// TwinCAT 3 PLC project PLC
// ProgramVersion: 3.1.4024.0
// libraries:
//   Tc2_Standard, * (Beckhoff Automation GmbH)
//   Tc2_System, * (Beckhoff Automation GmbH)
//   Tc3_Module, * (Beckhoff Automation GmbH)
// project tree:
//   / GlobalTextList.TcGTLO (not stored), PlcTask.TcTTO, VisualizationManager.TcVMO (not stored)
//   GVLs/ GVL.TcGVL (not stored)
//   POUs/ FB_VisuSim.TcPOU, MAIN.TcPOU (not stored), FB_StateMachine.TcPOU
//   VISUs/ Visu.TcVIS
// real-time tasks:
//   TASK PlcTask: cycle T#10ms, priority 20, ADS port 350
//   TASK VISU_TASK: cycle T#200000us, priority 30, ADS port 351

CONFIGURATION PLC
    RESOURCE PLC ON TwinCAT3
        TASK PlcTask(INTERVAL := T#10ms, PRIORITY := 20);
        PROGRAM MAIN WITH PlcTask : MAIN;
    END_RESOURCE
END_CONFIGURATION

// ---- POUs/FB_VisuSim.TcPOU
FUNCTION_BLOCK FB_VisuSim
VAR_INPUT
	bConveyor : BOOL;
END_VAR
VAR_OUTPUT
	bBottle : BOOL;
END_VAR
VAR
	fPos : REAL;
END_VAR

IF bConveyor THEN
	fPos := fPos + 0.1;
END_IF

IF fPos >= 100.0 THEN
	fPos := 0;
END_IF

bBottle := fPos >= 60.0 AND fPos <= 80.0;

END_FUNCTION_BLOCK

// ---- POUs/FB_StateMachine.TcPOU
(* -----------------------------------------------------------------------------
| This sample has been supplied by Beckhoff As-Is and is intended only as an   |
| example implementation. Functionality is not guaranteed.                     |
----------------------------------------------------------------------------- *)

FUNCTION_BLOCK FB_StateMachine
VAR_INPUT
	bStart : BOOL;
	bStop : BOOL;	
	bBottle : BOOL;				// fotocellula FC1	
END_VAR
VAR_OUTPUT
	bConveyor : BOOL;			// nastro trasportatore
	bWater : BOOL;				// riempimento acqua
	bMint : BOOL;				// riempimento menta	
	bCorking : BOOL;			// inserimento del tappo
END_VAR
VAR
	nStep : INT;
	
	fbTonBottle : TON;
	fbRtBottle : R_TRIG;
	
	fbTonStep2 : TON;
	fbTonStep3 : TON;
	fbTonStep4 : TON;
	fbTonStep5 : TON;
	fbTonStep6 : TON;
END_VAR

(* -----------------------------------------------------------------------------
| This sample has been supplied by Beckhoff As-Is and is intended only as an   |
| example implementation. Functionality is not guaranteed.                     |
----------------------------------------------------------------------------- *)

(* filtri *)
fbTonBottle(IN:= bBottle, PT:= T#500MS);		// filtro sensore presenza bottiglia

(* fronti *)
fbRtBottle(CLK:= fbTonBottle.Q);

(* tempo di permanenza negli step *)
fbTonStep2(IN:= nStep = 2, PT:= T#5S);			// tempo di riempimento acqua
fbTonStep3(IN:= nStep = 3, PT:= T#1S);			// tempo di riempimento menta
fbTonStep4(IN:= nStep = 4, PT:= T#1S);			// attesa prima di tappatura
fbTonStep5(IN:= nStep = 5, PT:= T#3S);			// tempo di tappatura
fbTonStep6(IN:= nStep = 6, PT:= T#1S);			// attesa dopo tappatura

CASE nStep OF
	0: (* macchina ferma *)
		bConveyor := FALSE;
		bWater := FALSE;
		bMint := FALSE;
		bCorking := FALSE;
		
		(* transition *)
		IF NOT bStop AND bStart THEN
			nStep := 1;
		END_IF
		
	1: (* avanzamento nastro *)
		bConveyor := TRUE;
		bWater := FALSE;
		bMint := FALSE;
		bCorking := FALSE;
		
		(* transition *)
		IF fbRtBottle.Q THEN
			nStep := 2;
		END_IF
		
	2: (* riempimento acqua *)
		bConveyor := FALSE;
		bWater := TRUE;
		bMint := FALSE;
		bCorking := FALSE;
		
		(* transition *)
		IF fbTonStep2.Q THEN
			nStep := 3;
		END_IF
		
	3: (* riempimento menta *)
		bConveyor := FALSE;
		bWater := FALSE;
		bMint := TRUE;
		bCorking := FALSE;
		
		(* transition *)
		IF fbTonStep3.Q THEN
			nStep := 4;
		END_IF
		
	4: (* attesa *)
		bConveyor := FALSE;
		bWater := FALSE;
		bMint := TRUE;
		bCorking := FALSE;
		
		(* transition *)
		IF fbTonStep4.Q THEN
			nStep := 5;
		END_IF
		
	5: (* tappatura *)
		bConveyor := FALSE;
		bWater := FALSE;
		bMint := FALSE;
		bCorking := TRUE;
		
		(* transition *)
		IF fbTonStep5.Q THEN
			nStep := 6;
		END_IF
		
	6: (* attesa *)
		bConveyor := FALSE;
		bWater := FALSE;
		bMint := FALSE;
		bCorking := FALSE;
		
		(* transition *)
		IF fbTonStep6.Q THEN
			nStep := 1;
		END_IF

END_CASE

END_FUNCTION_BLOCK

// ---- VISUs/Visu.TcVIS
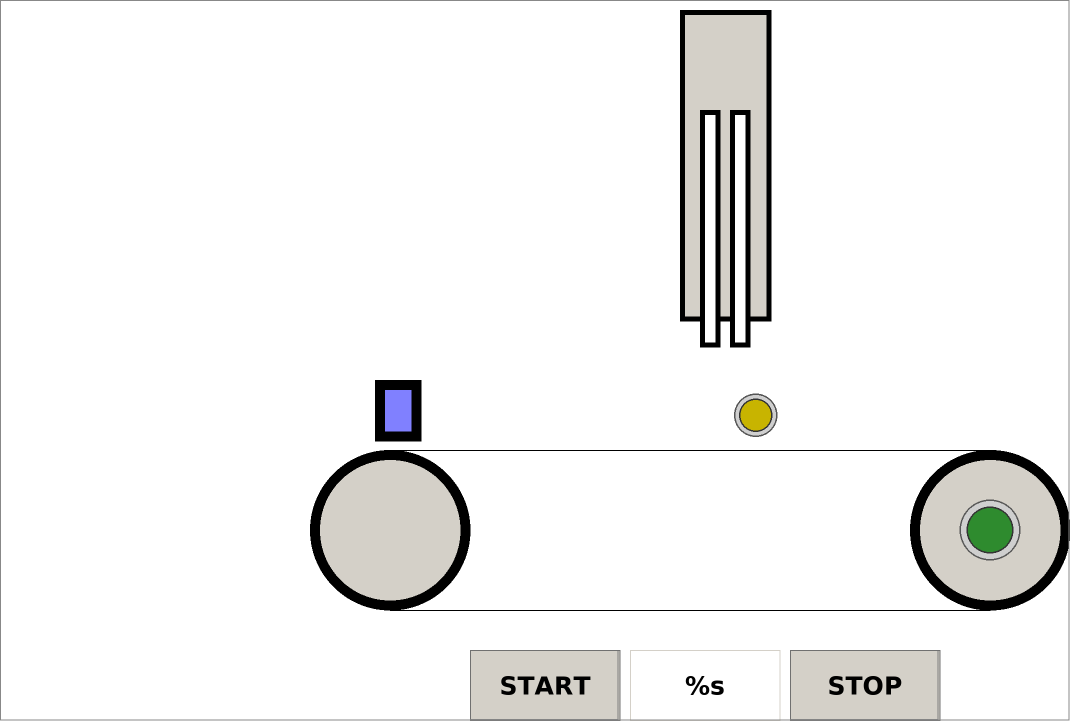
VISUALIZATION Visu  // 1070x721
    Rectangle (680,10 91x311), colour toggle: GVL.bCorking
        p2738717112: (TO_REAL(GVL.bCorking) * 50.0)
    Ellipse (310,450 160x160)
    Line (390,450) (990,450)
    Ellipse (910,450 160x160)
    Line (390,610) (990,610)
    Lamp1 (955,495 70x70), variable: GVL.bConveyor, style: Lamp-Lamp1-Green
    Rectangle (700,110 20x237), colour toggle: GVL.bWater
    Rectangle (730,110 20x237), colour toggle: GVL.bMint
    Button (470,650 150x71), "START"
        tap GVL.bStart
    Button (790,650 150x71), "STOP"
        tap GVL.bStop
    Textfield (630,650 150x71), "%s", text variable: MAIN.fbStateMachine.nStep
    Lamp1 (730,390 51x50), variable: GVL.bBottle, style: Lamp-Lamp1-Yellow
    RoundedRectangle (375,380 46x61)
        p3560616238: MAIN.fbVisuSim.fPos * 5.0
END_VISUALIZATION
